{attribute 'qualified_only'}
{attribute 'strict'}
TYPE E_FootpedalPos :
(
	eReverse2 	:= -2,
	eReverse1 	:= -1,
	eIdle		:= 0,
	eForward0	:= 1,
	eForward1	:= 2,
	eForward2	:= 3,
	eForward3	:= 4,
	eForward4	:= 5,
	eForward5	:= 6,
	eForward6	:= 7,
	eForward7	:= 8,
	eForward8	:= 9,
	eForward9	:= 10,
	eForward10	:= 11,
	eForward11	:= 12,
	eForward12	:= 13,
	eFalse			
) INT; 
END_TYPE
//  eReverse2 = '-2'
//  eReverse1 = '-1'

(* stored: Version 1.1.0.1, ProductVersion 3.1.4024.9
   EnumerationTextList E_FootpedalPos: Id {a45d04ff-12cb-4fd2-8aee-f6a35d915e0d} *)
